// Mitsubishi GX Works2 project: PLC_GROUP30   PLC: FX3G

// global labels: Global1
VAR_GLOBAL
  start AT X007 : BOOL;
  system_working AT Y007 : BOOL;
  end_day AT X005 : BOOL;
  start_melting AT X001 : BOOL;
END_VAR
VAR_GLOBAL CONSTANT
  chocolate_for_melting : REAL := 400.0;
END_VAR
VAR_GLOBAL
  chocolate_left AT D1100 : REAL;
  melting_light AT Y001 : BOOL;
  insert_chocolate AT D7000 : REAL;
  reched_temp_for_melting AT X002 : BOOL;
  start_casting AT X003 : BOOL;
END_VAR
VAR_GLOBAL CONSTANT
  casting_timer_time : INT := 40;
END_VAR
VAR_GLOBAL
  casting_timer AT TC0 : BOOL;
  insert_nuts AT D7002 : REAL;
  nuts_left AT D1102 : REAL;
  insert_pistachio AT D7004 : REAL;
  pistachio_left AT D1104 : REAL;
  qadaif_left AT D1106 : REAL;
  instert_qadaif AT D7006 : REAL;
  casting_light AT Y002 : BOOL;
  start_colling AT X006 : BOOL;
  cooling_timer AT TC2 : BOOL;
END_VAR
VAR_GLOBAL CONSTANT
  cooling_timer_time : INT := 30;
END_VAR
VAR_GLOBAL
  cooling_light AT Y006 : BOOL;
  casting_time_done AT TS0 : BOOL;
  cooling_timer_done AT TS2 : BOOL;
  analog_input_1 AT D8280 : INT;
END_VAR
VAR_GLOBAL CONSTANT
  analog_input_divide : REAL := 400;
END_VAR
VAR_GLOBAL
  user_chocolate_choice AT D1108 : REAL;
  start_chocolate_choise AT X004 : BOOL;
END_VAR
VAR_GLOBAL CONSTANT
  min_for_dubai : REAL := 5.0;
  max_for_dubai : REAL := 10.0;
  min_for_nuts : REAL;
END_VAR
VAR_GLOBAL
  chose_dubai AT M0 : BOOL;
  chose_nuts AT M1 : BOOL;
END_VAR
VAR_GLOBAL CONSTANT
  dubai_nuts_decrease : REAL := 20.0;
  dubai_pistachios_left : REAL := 120;
  dubai_qadaif_left : REAL := 60;
  nuts_nuts_decrease : REAL := 100;
  nuts_pistachios_left : REAL := 100;
END_VAR
VAR_GLOBAL
  filling_timer AT TC1 : BOOL;
END_VAR
VAR_GLOBAL CONSTANT
  filling_timer_time : INT := 50;
END_VAR
VAR_GLOBAL
  filling_timer_done AT TS1 : BOOL;
  blinking_demi AT M2 : BOOL;
  blinking_timer1 AT TC3 : BOOL;
END_VAR
VAR_GLOBAL CONSTANT
  blinking_time : INT := 10;
END_VAR
VAR_GLOBAL
  blinking_timer1_done AT TS3 : BOOL;
  blinking_light1 AT Y003 : BOOL;
  blinking_timer2 AT TC4 : BOOL;
  blinking_timer2_done AT TS4 : BOOL;
  blinking_light2 AT Y004 : BOOL;
  blinking_demi2 AT M3 : BOOL;
  can_start_casting AT M10 : BOOL;
  can_start_filling AT M11 : BOOL;
  can_start_cooling AT M12 : BOOL;
  boxing_of_piece AT X000 : BOOL;
  boxing_light AT Y005 : BOOL;
  boxing_counter AT CC0 : BOOL;
END_VAR
VAR_GLOBAL CONSTANT
  num_of_bars_in_box : INT := 4;
END_VAR
VAR_GLOBAL
  can_start_boxing AT M13 : BOOL;
  finished_boxing AT CS0 : BOOL;
END_VAR
VAR_GLOBAL CONSTANT
  zero : REAL;
  min_chocolate : REAL := 400;
  min_nuts : REAL := 100;
  min_pistachio : REAL := 120;
  min_qadaif : REAL := 60;
END_VAR
VAR_GLOBAL
  not_enough_materials AT M20 : BOOL;
END_VAR
VAR_GLOBAL CONSTANT
  one : INT := 1;
  analog_output_mul : INT := 40;
END_VAR
VAR_GLOBAL
  analog_output AT D8282 : INT;
  num_of_packages AT D1110 : REAL;
  reset_demi_lights AT M14 : BOOL;
END_VAR
VAR_GLOBAL CONSTANT
  big_number : REAL := 11;
END_VAR

// task Task_01 (event TRUE, interval 0, priority 31): POU_01

PROGRAM POU_01
(* structured ladder/FBD written out as ST: instructions are called as NAME(EN, inputs, outputs); _pN, _eN, _tN stand for wires *)
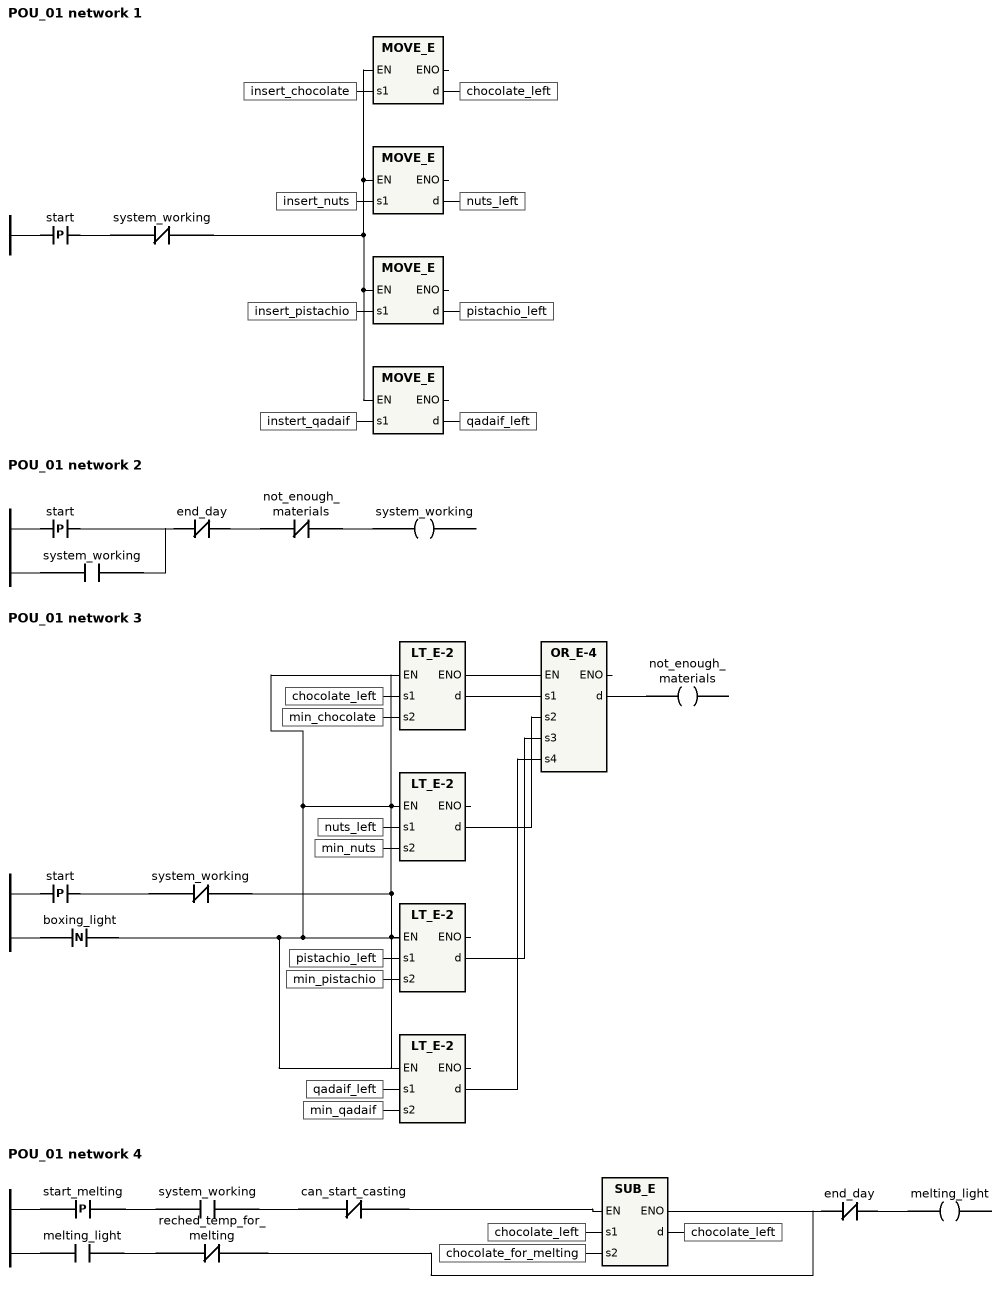
(* network 1 *)
_p1 := LDP(TRUE, start) AND NOT system_working;
MOVE_E(_p1, insert_chocolate, chocolate_left);
MOVE_E(_p1, insert_nuts, nuts_left);
MOVE_E(_p1, insert_pistachio, pistachio_left);
MOVE_E(_p1, instert_qadaif, qadaif_left);
(* network 2 *)
system_working := ((LDP(TRUE, start) OR system_working) AND NOT end_day) AND NOT not_enough_materials;
(* network 3 *)
_p1 := (LDP(TRUE, start) AND NOT system_working) OR LDF(TRUE, boxing_light);
_e3 := LT_E(_p1, chocolate_left, min_chocolate, _t2);
LT_E(_p1, nuts_left, min_nuts, _t4);
LT_E(_p1, pistachio_left, min_pistachio, _t5);
LT_E(_p1, qadaif_left, min_qadaif, _t6);
OR_E(_e3, _t2, _t4, _t5, _t6, _t7);
not_enough_materials := _t7;
(* network 4 *)
_e1 := SUB_E(LDP(TRUE, start_melting) AND system_working AND NOT can_start_casting, chocolate_left, chocolate_for_melting, chocolate_left);
melting_light := (_e1 OR (melting_light AND NOT reched_temp_for_melting)) AND NOT end_day;
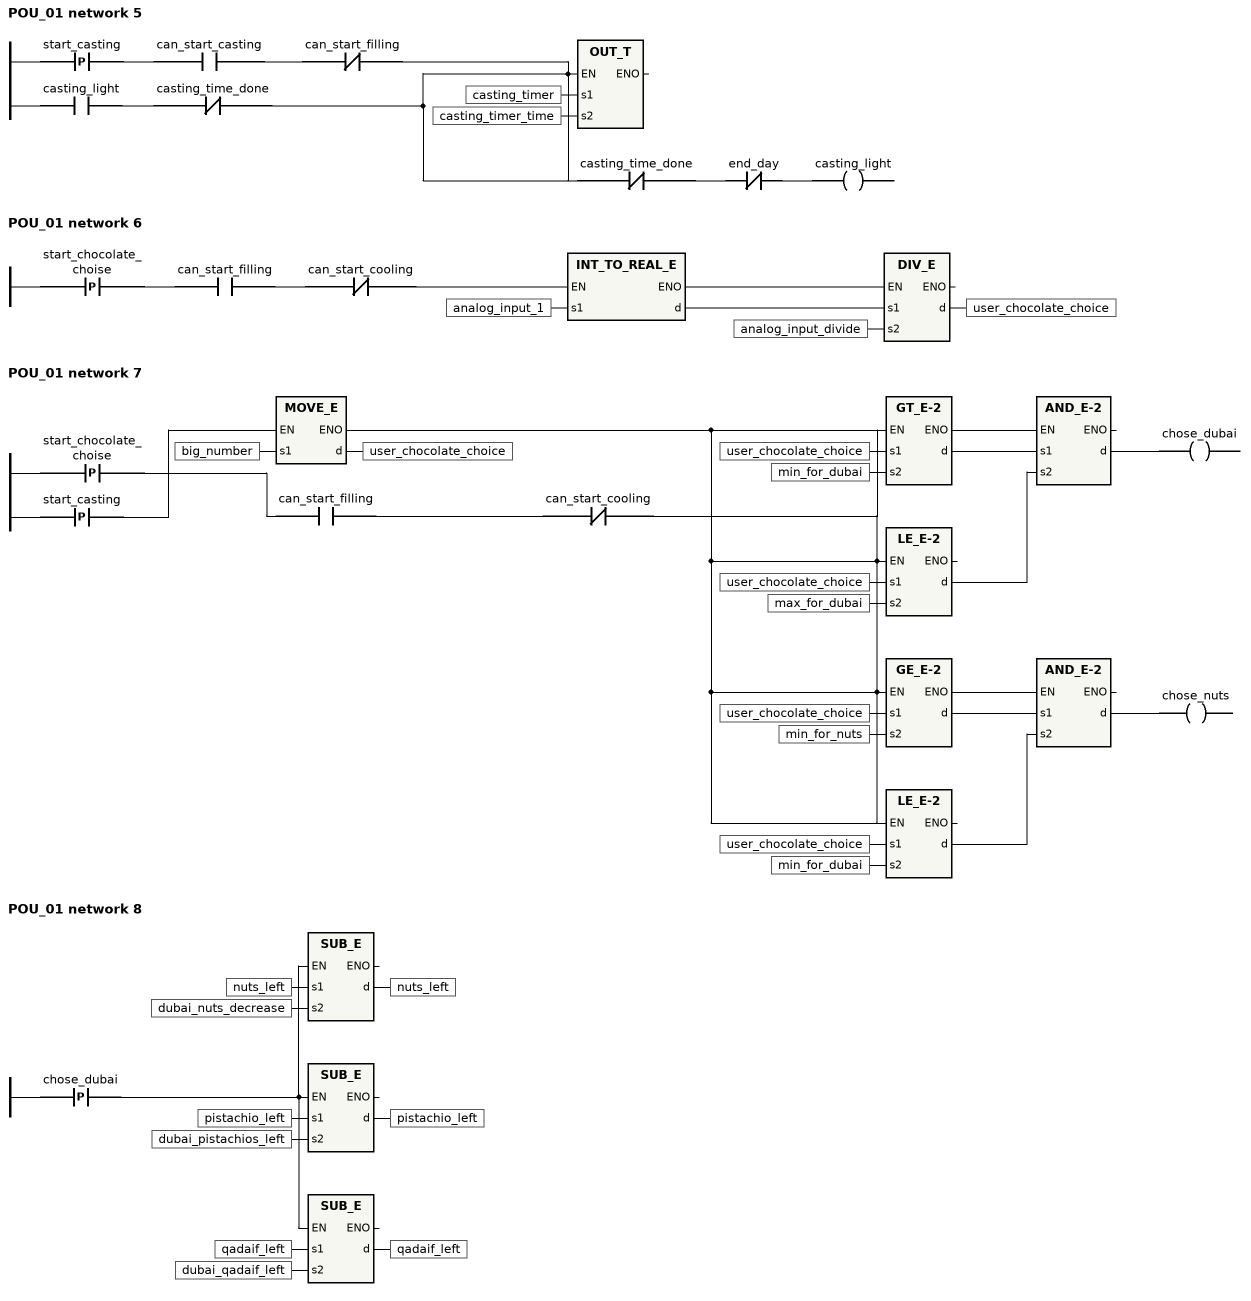
(* network 5 *)
_p1 := (LDP(TRUE, start_casting) AND can_start_casting AND NOT can_start_filling) OR (casting_light AND NOT casting_time_done);
casting_light := _p1 AND NOT casting_time_done AND NOT end_day;
OUT_T(_p1, casting_timer, casting_timer_time);
(* network 6 *)
_e2 := INT_TO_REAL_E(LDP(TRUE, start_chocolate_choise) AND can_start_filling AND NOT can_start_cooling, analog_input_1, _t1);
DIV_E(_e2, _t1, analog_input_divide, user_chocolate_choice);
(* network 7 *)
_e1 := MOVE_E(LDP(TRUE, start_casting), big_number, user_chocolate_choice);
_p2 := (LDP(TRUE, start_chocolate_choise) AND can_start_filling AND NOT can_start_cooling) OR _e1;
_e4 := GT_E(_p2, user_chocolate_choice, min_for_dubai, _t3);
LE_E(_p2, user_chocolate_choice, max_for_dubai, _t5);
AND_E(_e4, _t3, _t5, _t6);
chose_dubai := _t6;
_e8 := GE_E(_p2, user_chocolate_choice, min_for_nuts, _t7);
LE_E(_p2, user_chocolate_choice, min_for_dubai, _t9);
AND_E(_e8, _t7, _t9, _t10);
chose_nuts := _t10;
(* network 8 *)
_p1 := LDP(TRUE, chose_dubai);
SUB_E(_p1, nuts_left, dubai_nuts_decrease, nuts_left);
SUB_E(_p1, pistachio_left, dubai_pistachios_left, pistachio_left);
SUB_E(_p1, qadaif_left, dubai_qadaif_left, qadaif_left);
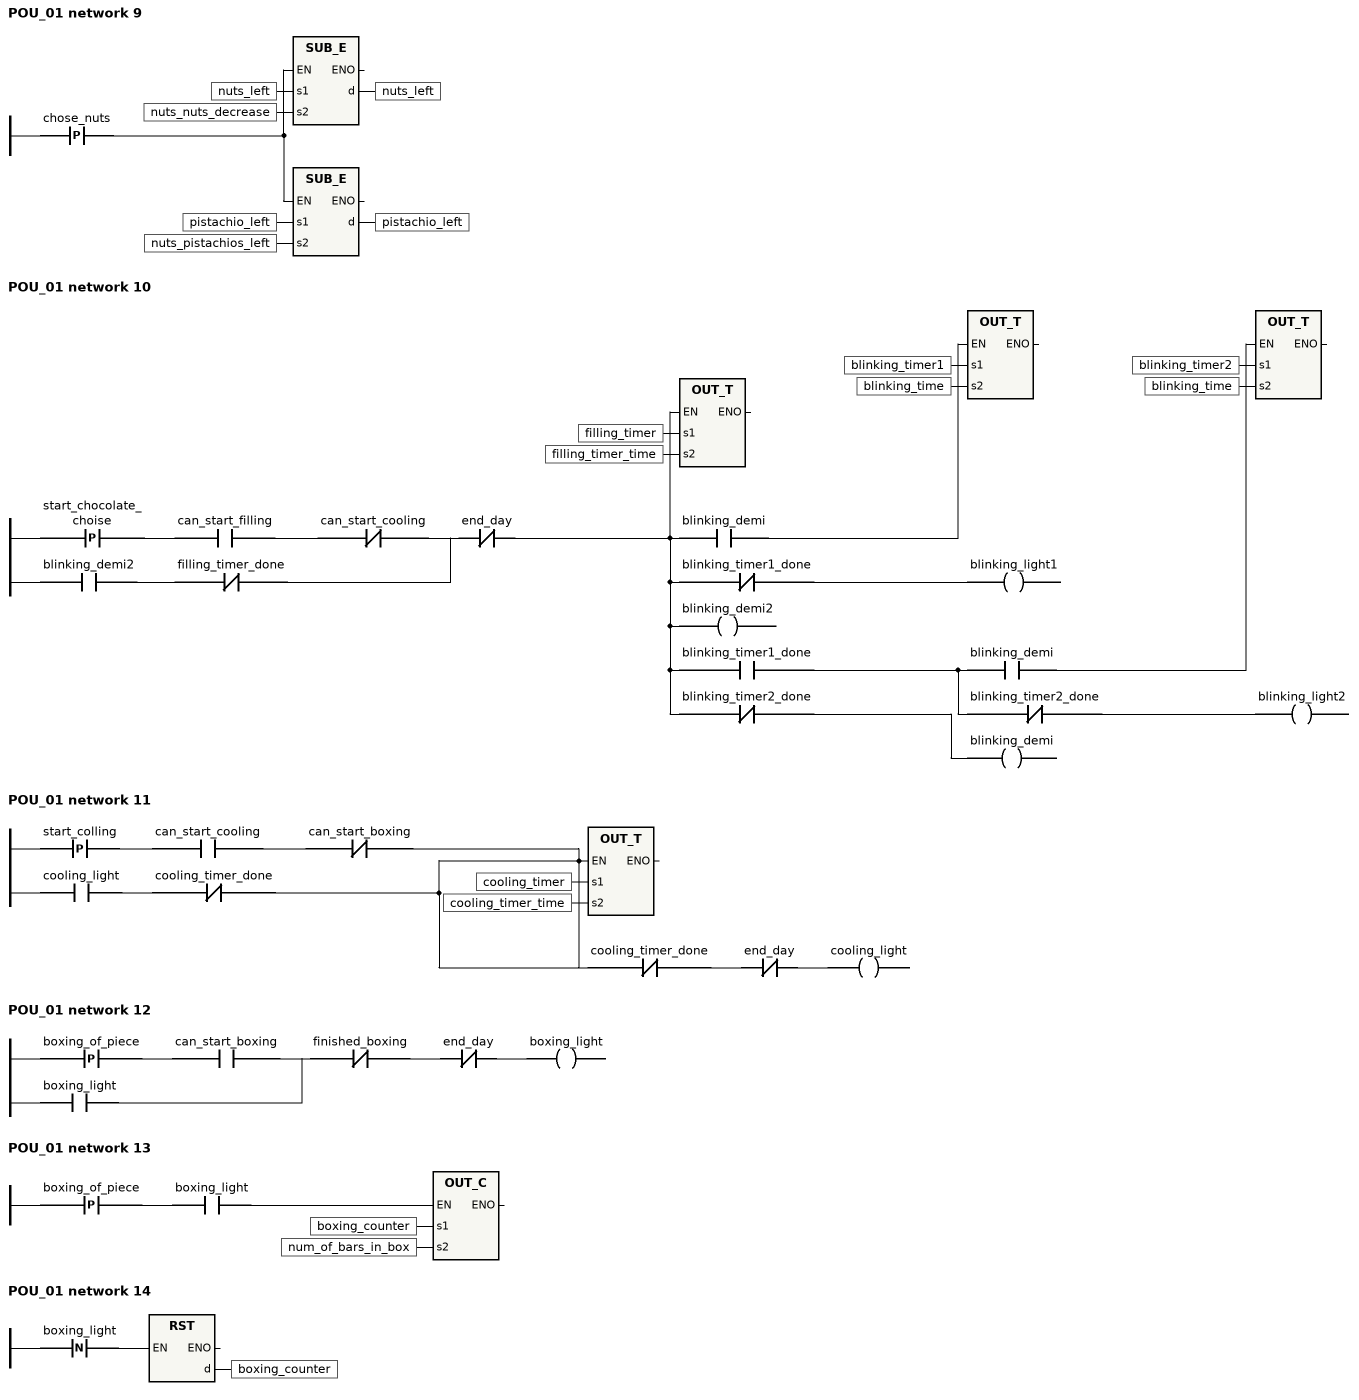
(* network 9 *)
_p1 := LDP(TRUE, chose_nuts);
SUB_E(_p1, nuts_left, nuts_nuts_decrease, nuts_left);
SUB_E(_p1, pistachio_left, nuts_pistachios_left, pistachio_left);
(* network 10 *)
_p1 := ((LDP(TRUE, start_chocolate_choise) AND can_start_filling AND NOT can_start_cooling) OR (blinking_demi2 AND NOT filling_timer_done)) AND NOT end_day;
OUT_T(_p1 AND blinking_demi, blinking_timer1, blinking_time);
blinking_light1 := _p1 AND NOT blinking_timer1_done;
OUT_T(_p1, filling_timer, filling_timer_time);
blinking_demi2 := _p1;
_p2 := _p1 AND blinking_timer1_done;
OUT_T(_p2 AND blinking_demi, blinking_timer2, blinking_time);
blinking_light2 := _p2 AND NOT blinking_timer2_done;
blinking_demi := _p1 AND NOT blinking_timer2_done;
(* network 11 *)
_p1 := (LDP(TRUE, start_colling) AND can_start_cooling AND NOT can_start_boxing) OR (cooling_light AND NOT cooling_timer_done);
cooling_light := _p1 AND NOT cooling_timer_done AND NOT end_day;
OUT_T(_p1, cooling_timer, cooling_timer_time);
(* network 12 *)
boxing_light := (((LDP(TRUE, boxing_of_piece) AND can_start_boxing) OR boxing_light) AND NOT finished_boxing) AND NOT end_day;
(* network 13 *)
OUT_C(LDP(TRUE, boxing_of_piece) AND boxing_light, boxing_counter, num_of_bars_in_box);
(* network 14 *)
RST(LDF(TRUE, boxing_light), boxing_counter);
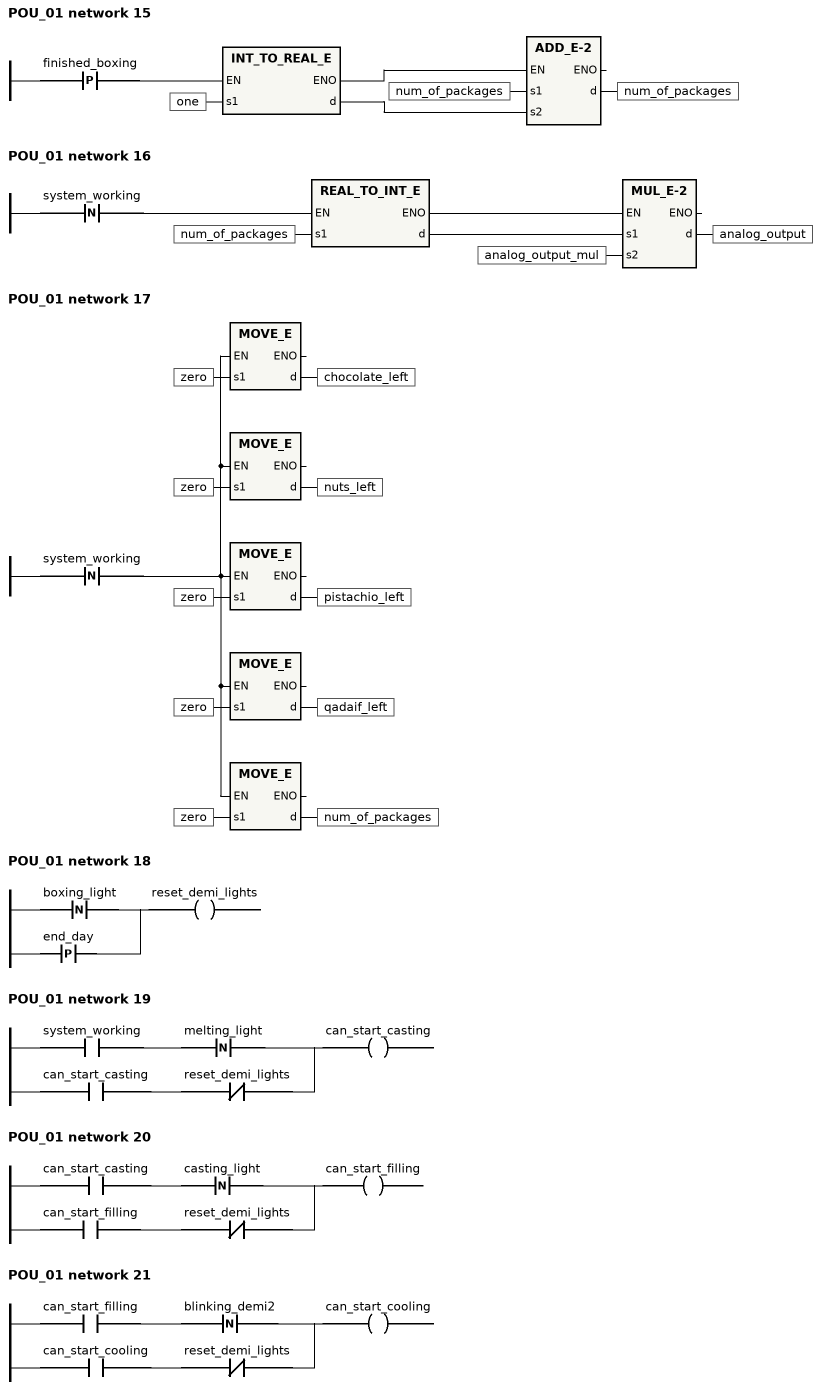
(* network 15 *)
_e2 := INT_TO_REAL_E(LDP(TRUE, finished_boxing), one, _t1);
ADD_E(_e2, num_of_packages, _t1, num_of_packages);
(* network 16 *)
_e2 := REAL_TO_INT_E(LDF(TRUE, system_working), num_of_packages, _t1);
MUL_E(_e2, _t1, analog_output_mul, analog_output);
(* network 17 *)
_p1 := LDF(TRUE, system_working);
MOVE_E(_p1, zero, chocolate_left);
MOVE_E(_p1, zero, nuts_left);
MOVE_E(_p1, zero, pistachio_left);
MOVE_E(_p1, zero, qadaif_left);
MOVE_E(_p1, zero, num_of_packages);
(* network 18 *)
reset_demi_lights := LDF(TRUE, boxing_light) OR LDP(TRUE, end_day);
(* network 19 *)
can_start_casting := (system_working AND LDF(TRUE, melting_light)) OR (can_start_casting AND NOT reset_demi_lights);
(* network 20 *)
can_start_filling := (can_start_casting AND LDF(TRUE, casting_light)) OR (can_start_filling AND NOT reset_demi_lights);
(* network 21 *)
can_start_cooling := (can_start_filling AND LDF(TRUE, blinking_demi2)) OR (can_start_cooling AND NOT reset_demi_lights);
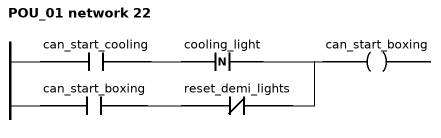
(* network 22 *)
can_start_boxing := (can_start_cooling AND LDF(TRUE, cooling_light)) OR (can_start_boxing AND NOT reset_demi_lights);
END_PROGRAM
